// SIMATIC S7-200 project (STEP 7-Micro/WIN), CPU 226 REL 02.00

SYMBOL_TABLE USR1
PV1              VW80
PV2              VW82
PV3              VW84
PV4              VW86
SV1              VW90
SV2              VW92
SV3              VW94
SV4              VW96
SET1             VW100
SET2             VW102
SET3             VW104
SET4             VW106
通讯开              V99.7
写                V99.6
读                V99.5
END_SYMBOL_TABLE

ORGANIZATION_BLOCK 主程序:OB1
TITLE=S7-200与富士PXR仪表自由通讯口协议通信
// 本程序基于西门子S7-200 PLC，通过RS485自由通讯口协议与富士PXR仪表实现工业烘箱温度监控与控制系统。系统通过PLC与富士PXR仪表的稳定通信，定期读取烘箱内多个区域的温度数据，并根据工艺需求向仪表写入温度设定值。
// 烘箱运行时，PLC每90毫秒轮询一次四个区域的温度传感器，确保所有区域温度数据实时更新。
// 富士PXR仪表连接四个温度传感器，分别监控烘箱内四个区域（例如顶部、底部、左侧、右侧）。
// 每次进行通信时，都需确保通信开关标志位已经被激活。
// 
// 初始化与富士PXR仪表的通信：
// 在做任何的操作之前，PLC会先检测通信就绪标志位，以此来检查PLC是否已经准备好与变频器进行通信。
// 富士 PXR 仪表在通信协议中规定，所有在通讯过程中所使用的符号，均需以ASCII格式方式来标识。
// 1）自由通讯口配置标志位设置为73，即自由通讯口协议采用9600波特率，8位字符，偶校验的模式。
// 2）自由通讯口的特性标志位为16#DC，即自由通讯口协议允许信息接收，并同时设置启始字符、不启用结束字符。
// 3）信息启始字符标志位为":"。空闲时间设置为5毫秒。接收超时设置为30毫秒。接收最大字符数设置为21。
// 
// 若通讯开关已打开，则启动90毫秒的通信定时器，开始通信流程。
// PLC通过通讯定时器分步与各传感器通信：通信定时器达到5毫秒时，在复位各个传感器的通信标志位。
// 通信定时器达到时，10毫秒、30毫秒、50毫秒、70毫秒时，分别一一激活第一、第二、第三、第四传感器通讯标志，逐个进行通信轮询。
// 在每个传感器的通讯轮询过程中，PLC根据从人机界面HMI设定的读取数据无效标志位和写操作许可标志位，决定是读取当前传感器的温度数值还是写入新设定值。若读取数据有效且不允许写，执行读操作。若允许写，无论读取数据是否有效，执行写操作。
// 在每次之前任何执行通信操作之前，需要激活通讯状态标志位，表示通信操作正在进行。
// PLC通过RCV指令接收仪表返回的数据，并使用中断INT1解码处理。
// 
// PLC向富士 PXR 仪表发送读取命令，让其返回指定的温度传感器的信息，并存储到指定的PLC变量当中。
// 富士 PXR 仪表在通信协议中规定，只能接受使用ASCII格式的数据，而PLC原来存储的信息都属于二进制数，所以在做数据交换操作之前，需要将数据转换为ASCII格式，才能开始交换数据。
// 进行发送操作的期间，应确认是否PLC与富士 PXR 仪表之间是有通讯请求信号，如果通讯请求信号被激活，才应开始完成任何通讯操作。
// 预设的读命令信息是一个仅有14字节长的数据帧，所以在获取预设的读命令赋值到XMT指令的发送缓冲区时，需要控制读取长度，避免出现数据溢出或数据混乱的情况。
// 在最终发送读命令之前，需要确认与目标的通讯链路是否正常，如果链路情况正常，才使用XMT指令发送读命令给PXR仪表，要求其返回该传感器的通讯数据，并存储到指定的PLC变量当中，否则重置通讯状态标志位，并置位错误信息标志返回。
// 在完成发送读命令后，PLC需要复位通讯状态标志位，结束本次读操作，为下一次的读/写操作做好准备。
// 
// PLC向富士PXR仪表发送写命令，将用户设定的温度值写入指定传感器，并接收反馈。
// 预设的写命令信息是一个18字节长的数据帧，所以在获取预设的写命令赋值到XMT缓冲区时，需要控制读取长度，避免出现数据溢出或数据混乱的情况。
// 在最终发送写命令之前，需要确认与目标的通讯链路是否正常，如果链路情况正常，才使用XMT指令发送读命令给PXR仪表，要求其返回该传感器的通讯数据，并存储到指定的PLC变量当中，否则重置通讯状态标志位，并置位错误信息标志返回。
// 在完成发送写命令后，PLC需要复位通讯状态标志位，结束本次读操作，为下一次的读/写操作做好准备。
// 中断INT1解码处理过程中每个步骤都需确保检查接收数据缓冲区长度为21个字节。
// 
BEGIN
Network 1
LD     SM0.1
CALL   自由口初始化:SBR3
Network 2
LD     SM0.0
CALL   通讯:SBR0
END_ORGANIZATION_BLOCK

SUBROUTINE_BLOCK 通讯:SBR0
TITLE=
BEGIN
Network 1
LDN    读:V99.5
AN     写:V99.6
O      写:V99.6
A      通讯开:V99.7
TON    T33, +90
Network 2
LDW=   T33, +5
R      V99.1, 4
Network 3
LDW=   T33, +10
S      V99.1, 1
R      SM87.7, 1
Network 4
LD     V99.1
LPS
A      写:V99.6
CALL   写命令:SBR2, +1, V99.1
LPP
AN     读:V99.5
AN     写:V99.6
CALL   读命令:SBR1, +1, V99.1
Network 5
LDW=   T33, +30
S      V99.2, 1
R      SM87.7, 1
Network 6
LD     V99.2
LPS
A      写:V99.6
CALL   写命令:SBR2, +2, V99.2
LPP
AN     读:V99.5
AN     写:V99.6
CALL   读命令:SBR1, +2, V99.2
Network 7
LDW=   T33, +50
S      V99.3, 1
Network 8
LD     V99.3
LPS
A      写:V99.6
CALL   写命令:SBR2, +3, V99.3
LPP
AN     读:V99.5
AN     写:V99.6
CALL   读命令:SBR1, +3, V99.3
Network 9
LDW=   T33, +70
S      V99.4, 1
R      SM87.7, 1
Network 10
LD     V99.4
LPS
A      写:V99.6
CALL   写命令:SBR2, +4, V99.4
LPP
AN     读:V99.5
AN     写:V99.6
CALL   读命令:SBR1, +4, V99.4
Network 11
LD     T33
LPS
A      写:V99.6
R      写:V99.6, 1
LPP
=      读:V99.5
Network 12
LD     SM4.5
RCV    VB50, 0
END_SUBROUTINE_BLOCK

SUBROUTINE_BLOCK 读命令:SBR1
TITLE=
// 
VAR_INPUT
Host:INT;	// LW0 
END_VAR
VAR_IN_OUT
Over:BOOL;	// L2.0 
END_VAR
BEGIN
Network 1
LD     SM0.0
MOVW   #Host:LW0, LW5
AENO
IBCD   LW5
AENO
HTA    LB6, VB3, 2
Network 2
LD     SM0.0
MOVW   +0, VW44
Network 3
LD     SM0.0
MOVD   &VB2, LD7
Network 4
LD     SM0.0
FOR    VW46, +1, +14
Network 5
LD     SM0.0
BTI    *LD7, LW3
AENO
+I     LW3, VW44
Network 6
LD     SM0.0
INCD   LD7
Network 7
NEXT
Network 8
LD     SM0.0
HTA    VB45, VB16, 2
Network 9
LD     SM4.5
XMT    VB0, 0
Network 10
LD     #Over:L2.0
R      #Over:L2.0, 1
END_SUBROUTINE_BLOCK

SUBROUTINE_BLOCK 写命令:SBR2
TITLE=
VAR_INPUT
Host:INT;	// LW0 
END_VAR
VAR_IN_OUT
Over:BOOL;	// L2.0 
END_VAR
BEGIN
Network 1
LD     SM0.0
MOVW   #Host:LW0, LW5
AENO
IBCD   LW5
AENO
HTA    LB6, VB23, 2
Network 2
LDW=   #Host:LW0, +1
MOVW   SET1:VW100, LW11
Network 3
LDW=   #Host:LW0, +2
MOVW   SET2:VW102, LW11
Network 4
LDW=   #Host:LW0, +3
MOVW   SET3:VW104, LW11
Network 5
LDW=   #Host:LW0, +4
MOVW   SET4:VW106, LW11
Network 6
LD     SM0.0
IBCD   LW11
AENO
HTA    LB11, VB34, 4
Network 7
LD     SM0.0
MOVW   +0, VW44
Network 8
LD     SM0.0
MOVD   &VB22, LD7
Network 9
LD     SM0.0
FOR    VW46, +1, +18
Network 10
LD     SM0.0
BTI    *LD7, LW3
AENO
+I     LW3, VW44
Network 11
LD     SM0.0
INCD   LD7
Network 12
NEXT
Network 13
LD     SM0.0
HTA    VB45, VB40, 2
Network 14
LD     SM4.5
XMT    VB20, 0
Network 15
LD     #Over:L2.0
R      #Over:L2.0, 1
END_SUBROUTINE_BLOCK

SUBROUTINE_BLOCK 自由口初始化:SBR3
TITLE=
BEGIN
Network 1
LD     SM0.0
MOVB   73, SMB30
MOVB   16#DC, SMB87
MOVB   16#3A, SMB88
MOVW   +5, SMW90
MOVW   +30, SMW92
MOVB   21, SMB94
Network 2
LD     SM0.0
ATCH   发送完成:INT0, 9
ATCH   解码:INT1, 23
ENI
Network 12 // 网络标题
// 网络注释
Network 22 // 网络标题
// 网络注释
END_SUBROUTINE_BLOCK

INTERRUPT_BLOCK 发送完成:INT0
TITLE=
BEGIN
Network 1
LD     SM0.0
S      SM87.7, 1
END_INTERRUPT_BLOCK

INTERRUPT_BLOCK 解码:INT1
TITLE=
BEGIN
Network 1
LDB=   VB50, 21
MOVB   VB50, VB400
AENO
ATH    VB58, VB72, 4
AENO
ATH    VB64, VB74, 4
Network 2
LDB=   VB50, 21
LPS
AB=    VB54, 16#31
MOVW   VW72, PV1:VW80
AENO
BCDI   PV1:VW80
AENO
MOVW   VW74, SV1:VW90
BCDI   SV1:VW90
LRD
AB=    VB54, 16#32
MOVW   VW72, PV2:VW82
AENO
BCDI   PV2:VW82
AENO
MOVW   VW74, SV2:VW92
BCDI   SV2:VW92
LRD
AB=    VB54, 16#33
MOVW   VW72, PV3:VW84
AENO
BCDI   PV3:VW84
AENO
MOVW   VW74, SV3:VW94
BCDI   SV3:VW94
LPP
AB=    VB200, 16#34
MOVW   VW72, PV4:VW86
AENO
BCDI   PV4:VW86
AENO
MOVW   VW74, SV4:VW96
BCDI   SV4:VW96
END_INTERRUPT_BLOCK

DATA_BLOCK_TAB USER1
BEGIN
VB0      17
VB1      16#3A
VB2      16#30
VB3      16#30
VB4      16#31
VB5      16#52
VB6      16#57
VB7      16#33
VB8      16#31
VB9      16#30
VB10     16#30
VB11     16#31
VB12     16#2C
VB13     16#32
VB14     16#D
VB15     16#A
VB16     16#42
VB17     16#34
VB20     21
VB21     16#3A
VB22     16#30
VB23     16#30
VB24     16#31
VB25     16#57
VB26     16#57
VB27     16#34
VB28     16#31
VB29     16#30
VB30     16#30
VB31     16#33
VB32     16#2C
VB33     16#30
VB34     16#30
VB35     16#30
VB36     16#35
VB37     16#34
VB38     16#D
VB39     16#A
VB40     16#36
VB41     16#32
VB99     2#10000000
END_DATA_BLOCK_TAB
